PROGRAM MAIN
VAR_OUTPUT
	currentTime : TIMESTRUCT;
END_VAR
VAR
	execute : BOOL;
	manualStep : BOOL := TRUE;
	manualSuction : BOOL := FALSE;
	stop : BOOL;
	
	moduleA22 : CarCorEx;
END_VAR
VAR
	getLocalTime : FB_LocalSystemTime;
	test : BOOL;
END_VAR

CallHardwareModules(); //start program with hardware call

SetupHardware();

callModules();

CallHardwareModules(); //end program with hardware call

//BundleToJson();

ACTION callModules:
getLocalTime(
	sNetID:= '', 
	bEnable:= TRUE, 
	dwCycle:= , 
	dwOpt:= , 
	tTimeout:= , 
	bValid=> , 
	systemTime=> currentTime, 
	tzID=> );

moduleA22(
	benderLeft:= benderA22Left, 
	robotLeft:= robot3, 
	robotRight:= robot4, 
	skidLeft:= skidA22Left, 
	skidRight:= skidA22Right, 
	magazineLeft:= magazineA22Left, 
	magazineRight:= magazineA22Right, 
	wrapper:= wrapperA22, 
	horizontalDriveLeft:= horizontalDriveA22Left, 
	horizontalDriveRight:= horizontalDriveA22Right, 
	verticalDriveLeft:= verticalDriveA22Left, 
	verticalDriveRight:= verticalDriveA22Right,  
	pistonBottom:= pistonA22Bottom, 
	suctionTopLeft:= suctionA22TopLeft, 
	suctionTopRight:= suctionA22TopRight, 
	suctionBottomLeft:= suctionA22BottomLeft, 
	suctionBottomRight:= suctionA22BottomRight, 
	suctionBottom:= suctionA22Bottom,
	pmlModeRequest=> , 
	pmlMode=> , 
	pmlState=> , 
	pmlCommand=> , 
	stop=> , 
	execute=> , 
	hold=> , 
	reset=> , 
	done=> , 
	error=> );
END_ACTION

END_PROGRAM

(* stored: Version 1.1.0.1, ProductVersion 3.1.4024.11
   POU MAIN: Id {bb23f57b-bfaa-4807-862f-695fb779bd1d}, SpecialFunc None
   Action callModules: Id {524a05bd-aa5d-4749-8232-9d95fc7a69c5} *)
